INTERFACE I_MotionTaskCollection EXTENDS I_TaskResult

METHOD AddTask
VAR_INPUT
	Task : I_MotionTask;
END_VAR
END_METHOD

{attribute 'monitoring' := 'call'}
PROPERTY ErrorTask : T_MaxString
GET
END_GET
END_PROPERTY

METHOD RemoveTaskByInstance
VAR_INPUT
	Task : I_MotionTask;
END_VAR
END_METHOD

END_INTERFACE

(* stored: Version 1.1.0.1, ProductVersion 3.1.4026.18
   Itf I_MotionTaskCollection: Id {5cef30fa-20ec-45a3-9abb-6d3952f0de91}
   Method AddTask: Id {2950274e-7e92-4b87-8014-c41a77a99a45}
   Property ErrorTask: Id {a06d0498-a6d5-4bd2-a621-0fd05c9b9e17}
   Get Get: Id {567eac01-b97a-4bff-8aae-681ceb940ee7}
   Method RemoveTaskByInstance: Id {7678a5bd-5735-492c-a995-a537ca3df1bd} *)
